Staubli VAL3: onF4Event.pgx

program onF4Event()
begin
  // look if the bButton is enable
  if bButton[3]
    // go to home


    ////    io:home=true
    ////    delay(0.5)
    ////    io:home=false

    if aioGet(MbAI_bMotorPowe)==1

      call use:timerDialog("Back To Home...",1)
      aioSet(MbAO_bAxis7Home,1)
      aioSet(MbAO_b7Axis,1)
      delay(0.5)
      wait(aioGet(MbAI_bHomeDone)==0 or isKeyPressed(255))
      if isKeyPressed(255)
        aioSet(MbAO_bStopMotor,1)
        delay(0.5)
        aioSet(MbAO_bStopMotor,0)
      endIf
      aioSet(MbAO_b7Axis,0)
    else
      if aioGet(MbAI_bMotorPowe)==0
        call use:timerDialog("7轴未上电",1)
      endIf

    endIf

    //
  endIf
end
